FUNCTION_BLOCK EffluentLogic (* CAT Function Block Type *)
  (* Standard: 61499-2 *)
  (* Version 0.0, 6/19/2026, Schneider Electric, template *)
  PACKAGE SE.Nereda;
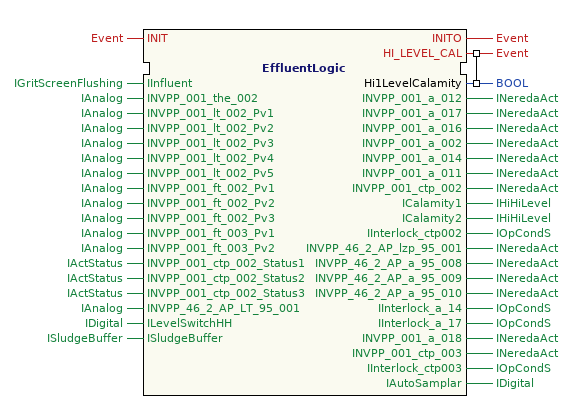
  EVENT_INPUT
    INIT;
  END_EVENT
  EVENT_OUTPUT
    INITO;
    HI_LEVEL_CAL WITH Hi1LevelCalamity; (* Input changed *)
  END_EVENT
  VAR_OUTPUT
    Hi1LevelCalamity : BOOL; (* Output value *)
  END_VAR
  SOCKETS
    IInfluent : IGritScreenFlushing;
    INVPP_001_the_002 : IAnalog;
  END_SOCKETS
  SOCKETS
    INVPP_001_lt_002_Pv1 : IAnalog;
    INVPP_001_lt_002_Pv2 : IAnalog;
    INVPP_001_lt_002_Pv3 : IAnalog;
    INVPP_001_lt_002_Pv4 : IAnalog;
    INVPP_001_lt_002_Pv5 : IAnalog;
    INVPP_001_ft_002_Pv1 : IAnalog;
    INVPP_001_ft_002_Pv2 : IAnalog;
    INVPP_001_ft_002_Pv3 : IAnalog;
    INVPP_001_ft_003_Pv1 : IAnalog;
    INVPP_001_ft_003_Pv2 : IAnalog; (* Process value (range considered) interface adapter *)
    INVPP_001_ctp_002_Status1 : IActStatus;
    INVPP_001_ctp_002_Status2 : IActStatus;
    INVPP_001_ctp_002_Status3 : IActStatus;
    INVPP_46_2_AP_LT_95_001 : IAnalog;
    ILevelSwitchHH : IDigital;
    ISludgeBuffer : ISludgeBuffer;
  END_SOCKETS
  PLUGS
    INVPP_001_a_012 : INeredaAct;
    INVPP_001_a_017 : INeredaAct;
    INVPP_001_a_016 : INeredaAct;
    INVPP_001_a_002 : INeredaAct;
    INVPP_001_a_014 : INeredaAct;
    INVPP_001_a_011 : INeredaAct;
    INVPP_001_ctp_002 : INeredaAct;
    ICalamity1 : IHiHiLevel;
    ICalamity2 : IHiHiLevel;
    IInterlock_ctp002 : IOpCondS; (* Condition summary chain output to downstream block *)
    INVPP_46_2_AP_lzp_95_001 : INeredaAct;
    INVPP_46_2_AP_a_95_008 : INeredaAct;
    INVPP_46_2_AP_a_95_009 : INeredaAct;
    INVPP_46_2_AP_a_95_010 : INeredaAct;
    IInterlock_a_14 : IOpCondS; (* Condition summary chain output to downstream block *)
    IInterlock_a_17 : IOpCondS; (* Condition summary chain output to downstream block *)
    INVPP_001_a_018 : INeredaAct;
    INVPP_001_ctp_003 : INeredaAct;
    IInterlock_ctp003 : IOpCondS; (* Condition summary chain output to downstream block *)
    IAutoSamplar : IDigital;
  END_PLUGS
  (* 01 - FUNCTIONNAL INPUT INTERFACE *)
  (* 00 - INITIALIZATION *)
  (* 05 - LOGIC *)
  (* 06 - HMI INTERFACE *)
  (* 03 - FIELD INTERFACE *)
  (* Flush Grit Screen Installation (Valve : NVPP_001_a_016 - NVPP_001_a_002) *)
  (* 02 - FUNCTIONNAL OUTPUT INTERFACE *)
  (* Flushing Manager *)
  (* Flush Grit Screens (Valve : NVPP_001_a_012) *)
  (* Flush Sludge Buffer (Valve : NVPP_001_a_017) *)
  (* Calamity *)
  (* Grit Screens Flushing Valve *)
  (* Sludge Buffer Flushing Valve *)
  (* Grit Screen Installation Flushing Valve *)
  (* Effluent Pump & Valves *)
  (* Calamity Pit *)
  (* To Final Treatment (To Nabehandeling) *)
  (* To Final Treatment (To Nabehandeling) *)
  (* Auto Samplar *)
  (* Auto Samplar *)
  (* Delayed Low Low Flow - Effluent Pump *)
  FBS
    FlushGritScreenInstallation : FlushGritScreenInstallation;
    FlushingManager : FlushingManager;
    Calamity : Calamity;
    IThis : EffluentLogic_HMI(QI := TRUE);
    ToFinalTreatment : ToFinalTreatment;
    AutoSamplar : AutoSamplar;
    DelayedLoLoFlowEffPump : EffLoLoFlowMng;
    FlushGritScreens : FlushGritScreens;
    FlushSludgeBuffer : FlushSludgeBuffer;
  END_FBS
  EVENT_CONNECTIONS
    INIT TO IThis.E36EC56CFB248E40;
    IThis.4BC7381B26F5C2BC TO FlushingManager.F242CF064A20C69F;
    FlushingManager.968F33EB7E7A6BCA TO Calamity.F242CF064A20C69F;
    Calamity.968F33EB7E7A6BCA TO ToFinalTreatment.F242CF064A20C69F;
    ToFinalTreatment.968F33EB7E7A6BCA TO FlushGritScreenInstallation.0681C0E37AE50C25;
    AutoSamplar.INITO TO INITO;
    FlushingManager.8BE5B82929E49AC6 TO Calamity.44F3C71D247046EA;
    IInfluent.9EB419218931A109 TO Calamity.D9A0D207EFE95E83;
    FlushSludgeBuffer.0CB0B64DB472C803 TO Calamity.0297B87FFCC4C5C4;
    Calamity.9897D33F12758EF0 TO HI_LEVEL_CAL;
    IInfluent.469E3B76B9D721DD TO FlushGritScreenInstallation.927E661A73225BAA;
    IInfluent.8B235293E5389BC7 TO FlushGritScreenInstallation.AF145550EB41F6EE;
    FlushGritScreenInstallation.0CB0B64DB472C803 TO IInfluent.727D767C86127C4D;
    IInfluent.8B235293E5389BC7 TO FlushGritScreens.AF145550EB41F6EE;
    INVPP_001_the_002.REQ TO IInfluent.0804B8CDC1B712F8;
    FlushSludgeBuffer.63C8A8D86F1B3EFF TO AutoSamplar.INIT;
    IInfluent.1F1020E82AE58441 TO AutoSamplar.INFLUENT_DRAIN_P;
    IInfluent.84E5BD043B0B9D2B TO AutoSamplar.PV_NVPP_FT_001;
    FlushGritScreenInstallation.367A5EB9A9086A3C TO IInfluent.9850048ED095E451;
    FlushGritScreenInstallation.63C8A8D86F1B3EFF TO FlushGritScreens.0681C0E37AE50C25;
    FlushGritScreens.63C8A8D86F1B3EFF TO FlushSludgeBuffer.0681C0E37AE50C25;
    IInfluent.469E3B76B9D721DD TO FlushGritScreens.927E661A73225BAA;
  END_CONNECTIONS
  DATA_CONNECTIONS
    FlushingManager.D6F2DD661B38D3B0 TO Calamity.2DDCBE290EE1C901;
    FlushingManager.DE7071ECCF601C73 TO Calamity.F069FF93C8395040;
    IInfluent.B8A74FB92C78BAA2 TO Calamity.E89E8852FE0B65F8;
    FlushSludgeBuffer.36BEB15804568122 TO Calamity.75A4C4FC23AB627D;
    Calamity.AC4FBD7D8FEA0F96 TO Hi1LevelCalamity;
    IInfluent.DB5751043930F3B0 TO FlushGritScreenInstallation.638C7342BE31DE35;
    IInfluent.917420DCD3928957 TO FlushGritScreenInstallation.F4AD8E05DB86547D;
    FlushGritScreenInstallation.36BEB15804568122 TO IInfluent.3A1846690B174C3E;
    IInfluent.917420DCD3928957 TO FlushGritScreens.F4AD8E05DB86547D;
    INVPP_001_the_002.Value TO IInfluent.F5105E8545B1ACE0;
    IInfluent.48F01954AB34CBCD TO AutoSamplar.InfluentDrainPump;
    IInfluent.1B5136012ECA25B4 TO AutoSamplar.Pv_NVPP_001_ft_001;
    FlushGritScreenInstallation.DDF028DDBF1BA194 TO IInfluent.9EB3C16A25E3E4D9;
    IInfluent.76B4FEAFDB90B7B7 TO FlushGritScreenInstallation.28FBEB94899DF3E5;
    IInfluent.DB5751043930F3B0 TO FlushGritScreens.638C7342BE31DE35;
    IInfluent.76B4FEAFDB90B7B7 TO FlushGritScreens.28FBEB94899DF3E5;
  END_CONNECTIONS
  ADAPTER_CONNECTIONS
    INVPP_001_ft_002_Pv2 TO FlushingManager.F282E8E66F83F2C8;
    INVPP_001_lt_002_Pv4 TO FlushingManager.28738E8901FA8ED4;
    INVPP_001_ft_002_Pv3 TO FlushingManager.8C1046847650A81C;
    FlushingManager.CADCAEF2966DB7AC TO INVPP_001_a_014;
    FlushingManager.D2F7FA931E666E8C TO INVPP_001_a_011;
    FlushingManager.3098C461BBAA5187 TO INVPP_001_ctp_002;
    FlushingManager.9CF466C1037A42DA TO FlushGritScreenInstallation.52A8D6A23243FFFE;
    FlushingManager.DB683E70D6D7177C TO FlushGritScreens.52A8D6A23243FFFE;
    FlushingManager.E6A9FE391D290C5E TO FlushSludgeBuffer.52A8D6A23243FFFE;
    FlushingManager.1945399653D28C5E TO IInterlock_ctp002;
    FlushingManager.61148D1353EE9735 TO IInterlock_a_14;
    INVPP_46_2_AP_LT_95_001 TO Calamity.3ED855F1C1BE1257;
    ILevelSwitchHH TO Calamity.D255585BBC8DADCD;
    ISludgeBuffer TO Calamity.F3A1B046E2898E98;
    Calamity.E05B50D2DCE5C504 TO ICalamity1;
    Calamity.91D044B45D837A64 TO ICalamity2;
    Calamity.BD4086BC52B92BB7 TO FlushingManager.E05B50D2DCE5C504;
    Calamity.FD2075D4A98928CD TO INVPP_46_2_AP_lzp_95_001;
    Calamity.5AC9F5AD8ED235A4 TO FlushSludgeBuffer.941D5B42A936047F;
    Calamity.3099FED8C7FE167A TO FlushSludgeBuffer.9371CBB2F0FE1F6B;
    Calamity.7C38394605374D59 TO INVPP_46_2_AP_a_95_008;
    Calamity.75A59846EA703249 TO INVPP_46_2_AP_a_95_009;
    Calamity.692DDFFCE9EA0F11 TO INVPP_46_2_AP_a_95_010;
    INVPP_001_lt_002_Pv5 TO ToFinalTreatment.28738E8901FA8ED4;
    INVPP_001_ft_003_Pv1 TO ToFinalTreatment.F282E8E66F83F2C8;
    INVPP_001_ft_003_Pv2 TO ToFinalTreatment.8C1046847650A81C;
    ToFinalTreatment.D2F7FA931E666E8C TO INVPP_001_a_018;
    ToFinalTreatment.3098C461BBAA5187 TO INVPP_001_ctp_003;
    ToFinalTreatment.1945399653D28C5E TO IInterlock_ctp003;
    INVPP_001_ft_002_Pv1 TO DelayedLoLoFlowEffPump.F7FFF31C0276695F;
    INVPP_001_lt_002_Pv3 TO FlushGritScreenInstallation.85FE606C922C82B2;
    INVPP_001_ctp_002_Status3 TO FlushGritScreenInstallation.458F685C95BC155A;
    FlushGritScreenInstallation.27D0C47F01DF2CD4 TO INVPP_001_a_016;
    FlushGritScreenInstallation.F7DB6D44A8BA20CC TO INVPP_001_a_002;
    INVPP_001_lt_002_Pv1 TO FlushGritScreens.85FE606C922C82B2;
    INVPP_001_ctp_002_Status1 TO FlushGritScreens.458F685C95BC155A;
    FlushGritScreens.F7DB6D44A8BA20CC TO INVPP_001_a_012;
    INVPP_001_lt_002_Pv2 TO FlushSludgeBuffer.85FE606C922C82B2;
    INVPP_001_ctp_002_Status2 TO FlushSludgeBuffer.458F685C95BC155A;
    FlushSludgeBuffer.F7DB6D44A8BA20CC TO INVPP_001_a_017;
    FlushSludgeBuffer.E28E60FFDFBEF43D TO IInterlock_a_17;
    AutoSamplar.423C240588CDA4C7 TO IAutoSamplar;
    DelayedLoLoFlowEffPump.EBD66E5BA2BD5929 TO FlushGritScreenInstallation.6E8E9C33428EDC72;
    DelayedLoLoFlowEffPump.F0A6495246D1224E TO FlushGritScreens.6E8E9C33428EDC72;
    DelayedLoLoFlowEffPump.24D55C4676B0D903 TO FlushSludgeBuffer.6E8E9C33428EDC72;
    FlushingManager.2C35D8FAC4D3EEBD TO DelayedLoLoFlowEffPump.78B0DAC8228293D0;
    FlushGritScreenInstallation.4DE6419011620A8C TO FlushGritScreens.8A147C4614F61E84;
    FlushGritScreenInstallation.2D599A4A0637E1A4 TO FlushSludgeBuffer.56D7A11F98C87B98;
    FlushGritScreens.938122B17C66C11D TO FlushSludgeBuffer.C252C4DA3115C78C;
  END_CONNECTIONS
END_FUNCTION_BLOCK
